{attribute 'linkalways'} 
{attribute 'no_explicit_call' := 'This FB is a CLASS and must be accessed using methods or properties'}
{attribute 'enable_dynamic_creation'}
FUNCTION_BLOCK Node_F_VN_MatchDescriptorsFlannLsh EXTENDS VisionNode
VAR
    ipQueryDescriptors : _ITcVnImage;
    ipTrainDescriptors : _ITcVnImage;
    ipMatches : _ITcVnContainer;
    hrPrev : _HRESULT(S_OK);
	hresult : _HRESULT(S_OK);
END_VAR

METHOD PUBLIC  Clone : I_Node
VAR
	pNode : POINTER TO Node_F_VN_MatchDescriptorsFlannLsh;
END_VAR
pNode := __NEW(Node_F_VN_MatchDescriptorsFlannLsh);
Clone := pNode^;
END_METHOD

METHOD FB_init : BOOL
VAR_INPUT
	bInitRetains : BOOL; // if TRUE, the retain variables are initialized (warm start / cold start)
	bInCopyCode : BOOL;  // if TRUE, the instance afterwards gets moved into the copy code (online change)
END_VAR
AddInput('ipQueryDescriptors', ipQueryDescriptors);
AddInput('ipTrainDescriptors', ipTrainDescriptors);
AddInput('hrPrev', hrPrev);
AddOutput('ipMatches', ipMatches);
AddOutput('hresult',hresult);
END_METHOD

METHOD PROTECTED OnExecute
hresult.Value := F_VN_MatchDescriptorsFlannLsh(
	ipQueryDescriptors := ipQueryDescriptors.Value,
    ipTrainDescriptors := ipTrainDescriptors.Value,
    ipMatches := ipMatches.Value,
	hrPrev:= hrPrev.Value);
END_METHOD

METHOD PUBLIC PreExecutionCheck
VAR_INPUT
	Check : I_PreExecutionChecks;
END_VAR
Check.IsTrue(ipQueryDescriptors.IsValid, 'ipQueryDescriptors must contain an image');
Check.IsTrue(ipTrainDescriptors.IsValid, 'ipTrainDescriptors must contain an image');
END_METHOD

END_FUNCTION_BLOCK

(* stored: Version 1.1.0.1, ProductVersion 3.1.4024.13
   POU Node_F_VN_MatchDescriptorsFlannLsh: Id {78bd0cb0-8ad9-0a41-06de-0751ab8313df}, SpecialFunc None
   Folder Constructor: Id {12082ac6-2fe9-0973-1414-3c63c5752e21}
   Method Clone: Id {eae8076c-d30f-01a7-09ab-fe1375f0066a}
   Method FB_init: Id {a93fedd6-de0e-0ff2-2e66-312b1ba9ffa3}
   Method OnExecute: Id {e23382b6-d7bd-06fc-34b9-fe57c28687b6}
   Method PreExecutionCheck: Id {f28bab46-47ed-008e-0e59-7a273bf4afcf} *)
